DATA_BLOCK "DB_Snd_BagsRep_T"
TITLE =%version: 0.02 % CN: 20
//History:
//This version  %created_by: nlhdl %
//              %date_created: maandag 7 december 2015 15:58:53 %
//              %release: VI_RAW/RA_Dev %
//
//Modification History:                                   By:    Date:     Rev:
//----------------------------------------------------  -------  --------  -----
//ra#9751: Add source files ECS-P to VI_RAW             nlHdL    14-12-15   0.02
//ra#9751: Add source files ECS-P to VI_RAW             nlHdL    07-12-15   0.02
//7632: Add TFC blocks to platform 4                    nlHdL    31-07-15   0.02
//20922: DB moved to NON RETAIN memory                  nlHdL    16-09-14   0.02
//18060: Update messages ID's for Vibes 3.2             nlHdL    01-04-14   0.01
//Initial Revision                                      nllHdL   20-02-14   0.01
//
FAMILY : VIBES
VERSION : 0.0
NON_RETAIN


  STRUCT
   Msgs : "UDT_Msg_BagsRep_T";
  END_STRUCT ;
BEGIN
END_DATA_BLOCK

